// TIA Portal V19 export
ORGANIZATION_BLOCK "MODBUS VFD"   // OB30, LAD, CyclicInterrupt
{ S7_Optimized_Access := 'TRUE' }
// stored: SetENOAutomatically false
   VAR_INPUT
      Initial_Call : Bool;   // Initial call of this OB
      Event_Count : Int;   // Events discarded
   END_VAR
   VAR_TEMP   // added for the SCL form of the ladder/FBD networks
      _w1 : Bool;
      _w2 : Bool;
   END_VAR
BEGIN

REGION Network 2: Slave 1 (SLAVE ID :- 1) WRITE
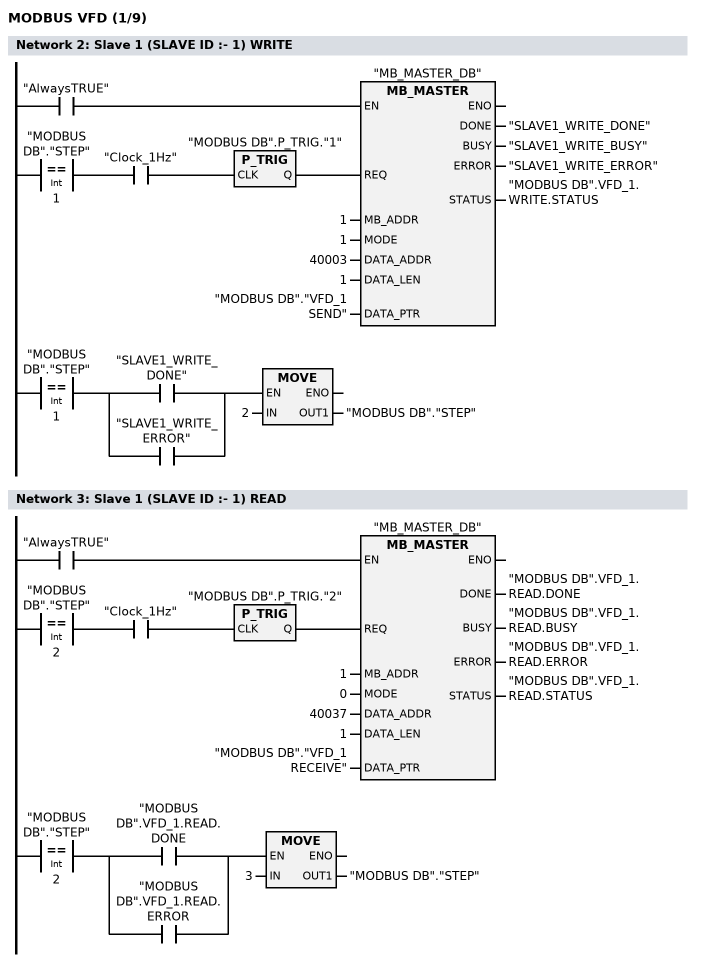
   RUNG wire#powerrail
      Contact( "AlwaysTRUE" )
      "MB_MASTER_DB".MB_MASTER(REQ := wire#w1, MB_ADDR := 1, MODE := 1, DATA_ADDR := 40003, DATA_LEN := 1, DATA_PTR := "MODBUS DB"."VFD_1 SEND", DONE => "SLAVE1_WRITE_DONE", BUSY => "SLAVE1_WRITE_BUSY", ERROR => "SLAVE1_WRITE_ERROR", STATUS => "MODBUS DB".VFD_1.WRITE.STATUS)
   END_RUNG
   RUNG wire#powerrail
      { S7_Templates := "SrcType := Int" } EQ_Contact(in1 := "MODBUS DB"."STEP", in2 := 1)
      Contact( "Clock_1Hz" )
      P_Trig( "MODBUS DB".P_TRIG."1" )
   END_RUNG wire#w1
   RUNG wire#powerrail
      { S7_Templates := "SrcType := Int" } EQ_Contact(in1 := "MODBUS DB"."STEP", in2 := 1)
      wire#w2
      Contact( "SLAVE1_WRITE_DONE" )
      wire#w3
      Move(in := 2, out1 => "MODBUS DB"."STEP")
   END_RUNG
   RUNG wire#w2
      Contact( "SLAVE1_WRITE_ERROR" )
   END_RUNG wire#w3
   // the same network as SCL:
   #_w1 := ("MODBUS DB"."STEP" = 1) AND "Clock_1Hz";
   #_w2 := #_w1 AND NOT "MODBUS DB".P_TRIG."1";   // rising edge
   "MODBUS DB".P_TRIG."1" := #_w1;
   IF "AlwaysTRUE" THEN
       "MB_MASTER_DB"(REQ := #_w2,   // MB_MASTER
                      MB_ADDR := 1,
                      MODE := 1,
                      DATA_ADDR := 40003,
                      DATA_LEN := 1,
                      DATA_PTR := "MODBUS DB"."VFD_1 SEND",
                      DONE => "SLAVE1_WRITE_DONE",
                      BUSY => "SLAVE1_WRITE_BUSY",
                      ERROR => "SLAVE1_WRITE_ERROR",
                      STATUS => "MODBUS DB".VFD_1.WRITE.STATUS);
   END_IF;
   IF ("MODBUS DB"."STEP" = 1) AND ("SLAVE1_WRITE_DONE" OR "SLAVE1_WRITE_ERROR") THEN
       "MODBUS DB"."STEP" := 2;
   END_IF;
END_REGION

REGION Network 3: Slave 1 (SLAVE ID :- 1) READ
   RUNG wire#powerrail
      Contact( "AlwaysTRUE" )
      "MB_MASTER_DB".MB_MASTER(REQ := wire#w1, MB_ADDR := 1, MODE := 0, DATA_ADDR := 40037, DATA_LEN := 1, DATA_PTR := "MODBUS DB"."VFD_1 RECEIVE", DONE => "MODBUS DB".VFD_1.READ.DONE, BUSY => "MODBUS DB".VFD_1.READ.BUSY, ERROR => "MODBUS DB".VFD_1.READ.ERROR, STATUS => "MODBUS DB".VFD_1.READ.STATUS)
   END_RUNG
   RUNG wire#powerrail
      { S7_Templates := "SrcType := Int" } EQ_Contact(in1 := "MODBUS DB"."STEP", in2 := 2)
      Contact( "Clock_1Hz" )
      P_Trig( "MODBUS DB".P_TRIG."2" )
   END_RUNG wire#w1
   RUNG wire#powerrail
      { S7_Templates := "SrcType := Int" } EQ_Contact(in1 := "MODBUS DB"."STEP", in2 := 2)
      wire#w2
      Contact( "MODBUS DB".VFD_1.READ.DONE )
      wire#w3
      Move(in := 3, out1 => "MODBUS DB"."STEP")
   END_RUNG
   RUNG wire#w2
      Contact( "MODBUS DB".VFD_1.READ.ERROR )
   END_RUNG wire#w3
   // the same network as SCL:
   #_w1 := ("MODBUS DB"."STEP" = 2) AND "Clock_1Hz";
   #_w2 := #_w1 AND NOT "MODBUS DB".P_TRIG."2";   // rising edge
   "MODBUS DB".P_TRIG."2" := #_w1;
   IF "AlwaysTRUE" THEN
       "MB_MASTER_DB"(REQ := #_w2,   // MB_MASTER
                      MB_ADDR := 1,
                      MODE := 0,
                      DATA_ADDR := 40037,
                      DATA_LEN := 1,
                      DATA_PTR := "MODBUS DB"."VFD_1 RECEIVE",
                      DONE => "MODBUS DB".VFD_1.READ.DONE,
                      BUSY => "MODBUS DB".VFD_1.READ.BUSY,
                      ERROR => "MODBUS DB".VFD_1.READ.ERROR,
                      STATUS => "MODBUS DB".VFD_1.READ.STATUS);
   END_IF;
   IF ("MODBUS DB"."STEP" = 2) AND ("MODBUS DB".VFD_1.READ.DONE OR "MODBUS DB".VFD_1.READ.ERROR) THEN
       "MODBUS DB"."STEP" := 3;
   END_IF;
END_REGION

REGION Network 4: Slave 2 (SLAVE ID :- 2) WRITE
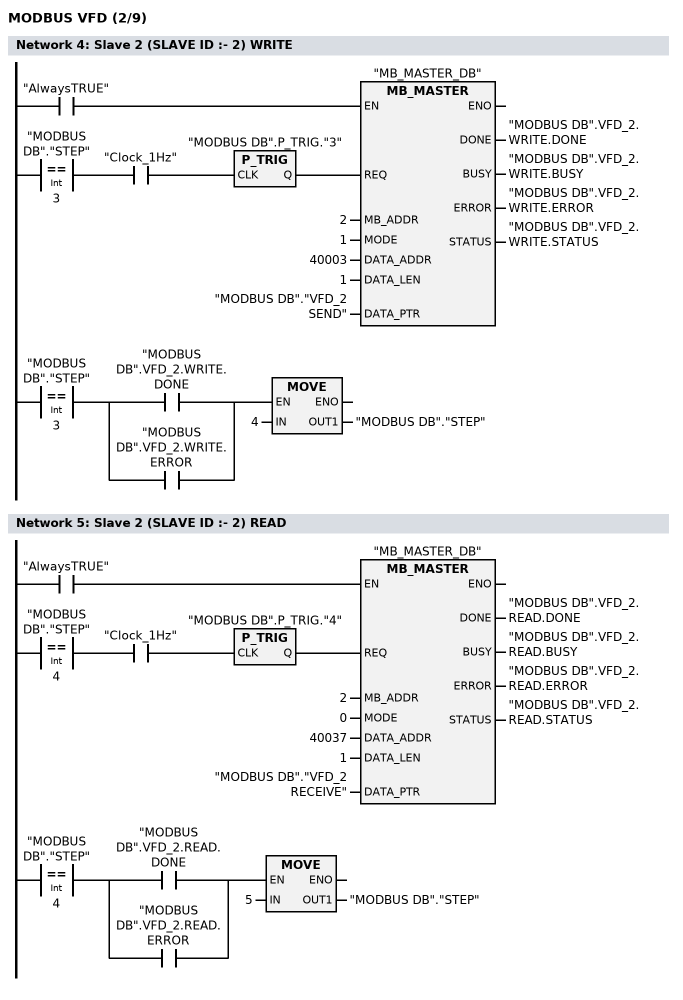
   RUNG wire#powerrail
      Contact( "AlwaysTRUE" )
      "MB_MASTER_DB".MB_MASTER(REQ := wire#w1, MB_ADDR := 2, MODE := 1, DATA_ADDR := 40003, DATA_LEN := 1, DATA_PTR := "MODBUS DB"."VFD_2 SEND", DONE => "MODBUS DB".VFD_2.WRITE.DONE, BUSY => "MODBUS DB".VFD_2.WRITE.BUSY, ERROR => "MODBUS DB".VFD_2.WRITE.ERROR, STATUS => "MODBUS DB".VFD_2.WRITE.STATUS)
   END_RUNG
   RUNG wire#powerrail
      { S7_Templates := "SrcType := Int" } EQ_Contact(in1 := "MODBUS DB"."STEP", in2 := 3)
      Contact( "Clock_1Hz" )
      P_Trig( "MODBUS DB".P_TRIG."3" )
   END_RUNG wire#w1
   RUNG wire#powerrail
      { S7_Templates := "SrcType := Int" } EQ_Contact(in1 := "MODBUS DB"."STEP", in2 := 3)
      wire#w2
      Contact( "MODBUS DB".VFD_2.WRITE.DONE )
      wire#w3
      Move(in := 4, out1 => "MODBUS DB"."STEP")
   END_RUNG
   RUNG wire#w2
      Contact( "MODBUS DB".VFD_2.WRITE.ERROR )
   END_RUNG wire#w3
   // the same network as SCL:
   #_w1 := ("MODBUS DB"."STEP" = 3) AND "Clock_1Hz";
   #_w2 := #_w1 AND NOT "MODBUS DB".P_TRIG."3";   // rising edge
   "MODBUS DB".P_TRIG."3" := #_w1;
   IF "AlwaysTRUE" THEN
       "MB_MASTER_DB"(REQ := #_w2,   // MB_MASTER
                      MB_ADDR := 2,
                      MODE := 1,
                      DATA_ADDR := 40003,
                      DATA_LEN := 1,
                      DATA_PTR := "MODBUS DB"."VFD_2 SEND",
                      DONE => "MODBUS DB".VFD_2.WRITE.DONE,
                      BUSY => "MODBUS DB".VFD_2.WRITE.BUSY,
                      ERROR => "MODBUS DB".VFD_2.WRITE.ERROR,
                      STATUS => "MODBUS DB".VFD_2.WRITE.STATUS);
   END_IF;
   IF ("MODBUS DB"."STEP" = 3) AND ("MODBUS DB".VFD_2.WRITE.DONE OR "MODBUS DB".VFD_2.WRITE.ERROR) THEN
       "MODBUS DB"."STEP" := 4;
   END_IF;
END_REGION

REGION Network 5: Slave 2 (SLAVE ID :- 2) READ
   RUNG wire#powerrail
      Contact( "AlwaysTRUE" )
      "MB_MASTER_DB".MB_MASTER(REQ := wire#w1, MB_ADDR := 2, MODE := 0, DATA_ADDR := 40037, DATA_LEN := 1, DATA_PTR := "MODBUS DB"."VFD_2 RECEIVE", DONE => "MODBUS DB".VFD_2.READ.DONE, BUSY => "MODBUS DB".VFD_2.READ.BUSY, ERROR => "MODBUS DB".VFD_2.READ.ERROR, STATUS => "MODBUS DB".VFD_2.READ.STATUS)
   END_RUNG
   RUNG wire#powerrail
      { S7_Templates := "SrcType := Int" } EQ_Contact(in1 := "MODBUS DB"."STEP", in2 := 4)
      Contact( "Clock_1Hz" )
      P_Trig( "MODBUS DB".P_TRIG."4" )
   END_RUNG wire#w1
   RUNG wire#powerrail
      { S7_Templates := "SrcType := Int" } EQ_Contact(in1 := "MODBUS DB"."STEP", in2 := 4)
      wire#w2
      Contact( "MODBUS DB".VFD_2.READ.DONE )
      wire#w3
      Move(in := 5, out1 => "MODBUS DB"."STEP")
   END_RUNG
   RUNG wire#w2
      Contact( "MODBUS DB".VFD_2.READ.ERROR )
   END_RUNG wire#w3
   // the same network as SCL:
   #_w1 := ("MODBUS DB"."STEP" = 4) AND "Clock_1Hz";
   #_w2 := #_w1 AND NOT "MODBUS DB".P_TRIG."4";   // rising edge
   "MODBUS DB".P_TRIG."4" := #_w1;
   IF "AlwaysTRUE" THEN
       "MB_MASTER_DB"(REQ := #_w2,   // MB_MASTER
                      MB_ADDR := 2,
                      MODE := 0,
                      DATA_ADDR := 40037,
                      DATA_LEN := 1,
                      DATA_PTR := "MODBUS DB"."VFD_2 RECEIVE",
                      DONE => "MODBUS DB".VFD_2.READ.DONE,
                      BUSY => "MODBUS DB".VFD_2.READ.BUSY,
                      ERROR => "MODBUS DB".VFD_2.READ.ERROR,
                      STATUS => "MODBUS DB".VFD_2.READ.STATUS);
   END_IF;
   IF ("MODBUS DB"."STEP" = 4) AND ("MODBUS DB".VFD_2.READ.DONE OR "MODBUS DB".VFD_2.READ.ERROR) THEN
       "MODBUS DB"."STEP" := 5;
   END_IF;
END_REGION

REGION Network 6: Slave 3 (SLAVE ID :- 3) WRITE
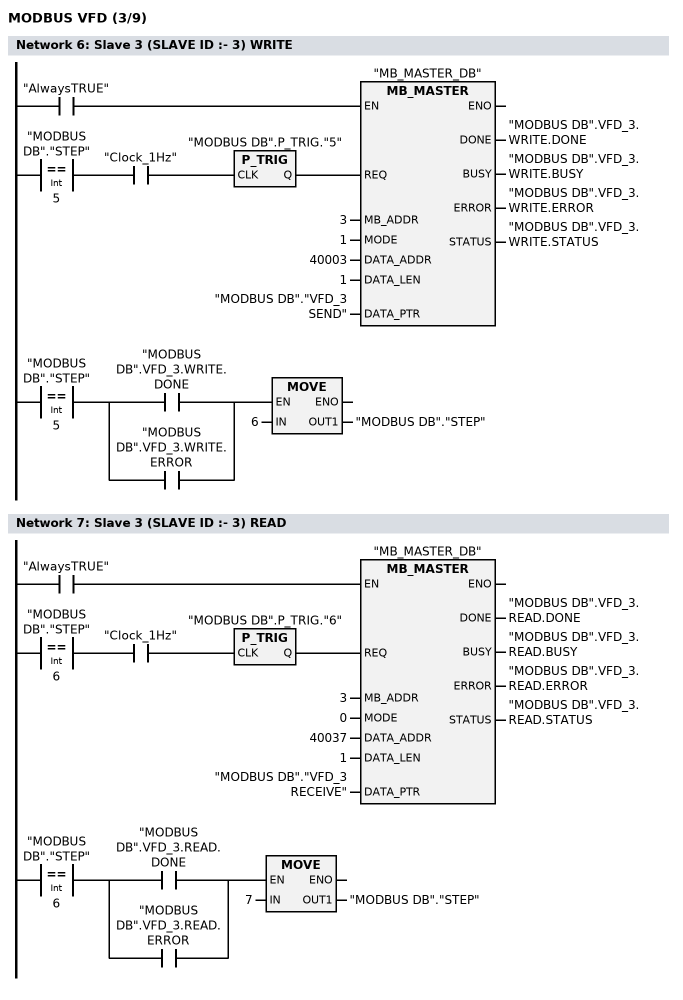
   RUNG wire#powerrail
      Contact( "AlwaysTRUE" )
      "MB_MASTER_DB".MB_MASTER(REQ := wire#w1, MB_ADDR := 3, MODE := 1, DATA_ADDR := 40003, DATA_LEN := 1, DATA_PTR := "MODBUS DB"."VFD_3 SEND", DONE => "MODBUS DB".VFD_3.WRITE.DONE, BUSY => "MODBUS DB".VFD_3.WRITE.BUSY, ERROR => "MODBUS DB".VFD_3.WRITE.ERROR, STATUS => "MODBUS DB".VFD_3.WRITE.STATUS)
   END_RUNG
   RUNG wire#powerrail
      { S7_Templates := "SrcType := Int" } EQ_Contact(in1 := "MODBUS DB"."STEP", in2 := 5)
      Contact( "Clock_1Hz" )
      P_Trig( "MODBUS DB".P_TRIG."5" )
   END_RUNG wire#w1
   RUNG wire#powerrail
      { S7_Templates := "SrcType := Int" } EQ_Contact(in1 := "MODBUS DB"."STEP", in2 := 5)
      wire#w2
      Contact( "MODBUS DB".VFD_3.WRITE.DONE )
      wire#w3
      Move(in := 6, out1 => "MODBUS DB"."STEP")
   END_RUNG
   RUNG wire#w2
      Contact( "MODBUS DB".VFD_3.WRITE.ERROR )
   END_RUNG wire#w3
   // the same network as SCL:
   #_w1 := ("MODBUS DB"."STEP" = 5) AND "Clock_1Hz";
   #_w2 := #_w1 AND NOT "MODBUS DB".P_TRIG."5";   // rising edge
   "MODBUS DB".P_TRIG."5" := #_w1;
   IF "AlwaysTRUE" THEN
       "MB_MASTER_DB"(REQ := #_w2,   // MB_MASTER
                      MB_ADDR := 3,
                      MODE := 1,
                      DATA_ADDR := 40003,
                      DATA_LEN := 1,
                      DATA_PTR := "MODBUS DB"."VFD_3 SEND",
                      DONE => "MODBUS DB".VFD_3.WRITE.DONE,
                      BUSY => "MODBUS DB".VFD_3.WRITE.BUSY,
                      ERROR => "MODBUS DB".VFD_3.WRITE.ERROR,
                      STATUS => "MODBUS DB".VFD_3.WRITE.STATUS);
   END_IF;
   IF ("MODBUS DB"."STEP" = 5) AND ("MODBUS DB".VFD_3.WRITE.DONE OR "MODBUS DB".VFD_3.WRITE.ERROR) THEN
       "MODBUS DB"."STEP" := 6;
   END_IF;
END_REGION

REGION Network 7: Slave 3 (SLAVE ID :- 3) READ
   RUNG wire#powerrail
      Contact( "AlwaysTRUE" )
      "MB_MASTER_DB".MB_MASTER(REQ := wire#w1, MB_ADDR := 3, MODE := 0, DATA_ADDR := 40037, DATA_LEN := 1, DATA_PTR := "MODBUS DB"."VFD_3 RECEIVE", DONE => "MODBUS DB".VFD_3.READ.DONE, BUSY => "MODBUS DB".VFD_3.READ.BUSY, ERROR => "MODBUS DB".VFD_3.READ.ERROR, STATUS => "MODBUS DB".VFD_3.READ.STATUS)
   END_RUNG
   RUNG wire#powerrail
      { S7_Templates := "SrcType := Int" } EQ_Contact(in1 := "MODBUS DB"."STEP", in2 := 6)
      Contact( "Clock_1Hz" )
      P_Trig( "MODBUS DB".P_TRIG."6" )
   END_RUNG wire#w1
   RUNG wire#powerrail
      { S7_Templates := "SrcType := Int" } EQ_Contact(in1 := "MODBUS DB"."STEP", in2 := 6)
      wire#w2
      Contact( "MODBUS DB".VFD_3.READ.DONE )
      wire#w3
      Move(in := 7, out1 => "MODBUS DB"."STEP")
   END_RUNG
   RUNG wire#w2
      Contact( "MODBUS DB".VFD_3.READ.ERROR )
   END_RUNG wire#w3
   // the same network as SCL:
   #_w1 := ("MODBUS DB"."STEP" = 6) AND "Clock_1Hz";
   #_w2 := #_w1 AND NOT "MODBUS DB".P_TRIG."6";   // rising edge
   "MODBUS DB".P_TRIG."6" := #_w1;
   IF "AlwaysTRUE" THEN
       "MB_MASTER_DB"(REQ := #_w2,   // MB_MASTER
                      MB_ADDR := 3,
                      MODE := 0,
                      DATA_ADDR := 40037,
                      DATA_LEN := 1,
                      DATA_PTR := "MODBUS DB"."VFD_3 RECEIVE",
                      DONE => "MODBUS DB".VFD_3.READ.DONE,
                      BUSY => "MODBUS DB".VFD_3.READ.BUSY,
                      ERROR => "MODBUS DB".VFD_3.READ.ERROR,
                      STATUS => "MODBUS DB".VFD_3.READ.STATUS);
   END_IF;
   IF ("MODBUS DB"."STEP" = 6) AND ("MODBUS DB".VFD_3.READ.DONE OR "MODBUS DB".VFD_3.READ.ERROR) THEN
       "MODBUS DB"."STEP" := 7;
   END_IF;
END_REGION

REGION Network 8: Slave 4 (SLAVE ID :- 4) WRITE
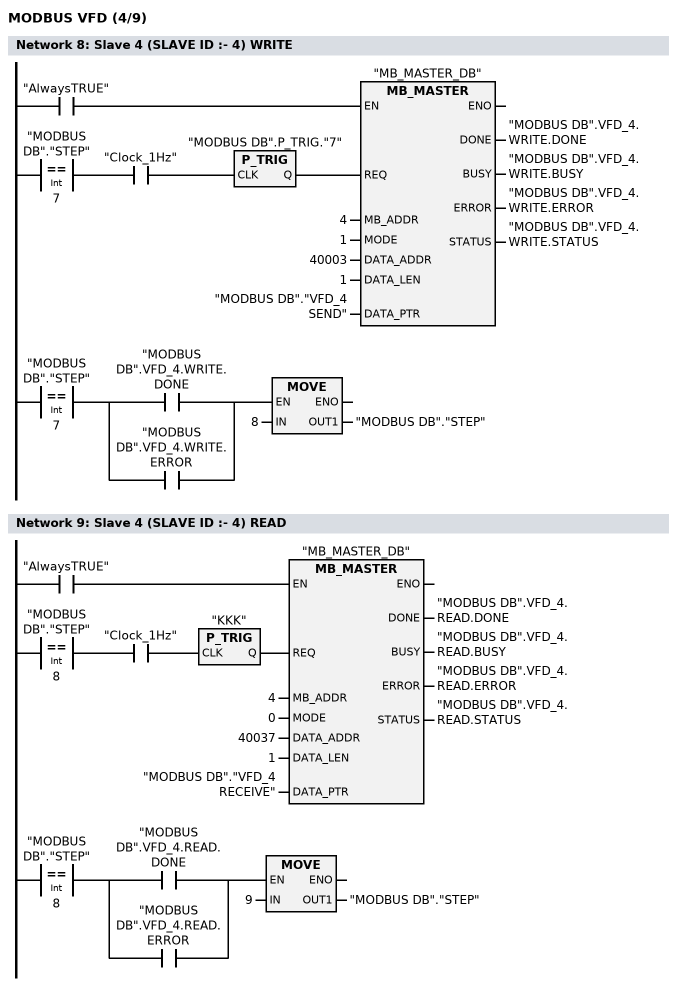
   RUNG wire#powerrail
      Contact( "AlwaysTRUE" )
      "MB_MASTER_DB".MB_MASTER(REQ := wire#w1, MB_ADDR := 4, MODE := 1, DATA_ADDR := 40003, DATA_LEN := 1, DATA_PTR := "MODBUS DB"."VFD_4 SEND", DONE => "MODBUS DB".VFD_4.WRITE.DONE, BUSY => "MODBUS DB".VFD_4.WRITE.BUSY, ERROR => "MODBUS DB".VFD_4.WRITE.ERROR, STATUS => "MODBUS DB".VFD_4.WRITE.STATUS)
   END_RUNG
   RUNG wire#powerrail
      { S7_Templates := "SrcType := Int" } EQ_Contact(in1 := "MODBUS DB"."STEP", in2 := 7)
      Contact( "Clock_1Hz" )
      P_Trig( "MODBUS DB".P_TRIG."7" )
   END_RUNG wire#w1
   RUNG wire#powerrail
      { S7_Templates := "SrcType := Int" } EQ_Contact(in1 := "MODBUS DB"."STEP", in2 := 7)
      wire#w2
      Contact( "MODBUS DB".VFD_4.WRITE.DONE )
      wire#w3
      Move(in := 8, out1 => "MODBUS DB"."STEP")
   END_RUNG
   RUNG wire#w2
      Contact( "MODBUS DB".VFD_4.WRITE.ERROR )
   END_RUNG wire#w3
   // the same network as SCL:
   #_w1 := ("MODBUS DB"."STEP" = 7) AND "Clock_1Hz";
   #_w2 := #_w1 AND NOT "MODBUS DB".P_TRIG."7";   // rising edge
   "MODBUS DB".P_TRIG."7" := #_w1;
   IF "AlwaysTRUE" THEN
       "MB_MASTER_DB"(REQ := #_w2,   // MB_MASTER
                      MB_ADDR := 4,
                      MODE := 1,
                      DATA_ADDR := 40003,
                      DATA_LEN := 1,
                      DATA_PTR := "MODBUS DB"."VFD_4 SEND",
                      DONE => "MODBUS DB".VFD_4.WRITE.DONE,
                      BUSY => "MODBUS DB".VFD_4.WRITE.BUSY,
                      ERROR => "MODBUS DB".VFD_4.WRITE.ERROR,
                      STATUS => "MODBUS DB".VFD_4.WRITE.STATUS);
   END_IF;
   IF ("MODBUS DB"."STEP" = 7) AND ("MODBUS DB".VFD_4.WRITE.DONE OR "MODBUS DB".VFD_4.WRITE.ERROR) THEN
       "MODBUS DB"."STEP" := 8;
   END_IF;
END_REGION

REGION Network 9: Slave 4 (SLAVE ID :- 4) READ
   RUNG wire#powerrail
      Contact( "AlwaysTRUE" )
      "MB_MASTER_DB".MB_MASTER(REQ := wire#w1, MB_ADDR := 4, MODE := 0, DATA_ADDR := 40037, DATA_LEN := 1, DATA_PTR := "MODBUS DB"."VFD_4 RECEIVE", DONE => "MODBUS DB".VFD_4.READ.DONE, BUSY => "MODBUS DB".VFD_4.READ.BUSY, ERROR => "MODBUS DB".VFD_4.READ.ERROR, STATUS => "MODBUS DB".VFD_4.READ.STATUS)
   END_RUNG
   RUNG wire#powerrail
      { S7_Templates := "SrcType := Int" } EQ_Contact(in1 := "MODBUS DB"."STEP", in2 := 8)
      Contact( "Clock_1Hz" )
      P_Trig( "KKK" )
   END_RUNG wire#w1
   RUNG wire#powerrail
      { S7_Templates := "SrcType := Int" } EQ_Contact(in1 := "MODBUS DB"."STEP", in2 := 8)
      wire#w2
      Contact( "MODBUS DB".VFD_4.READ.DONE )
      wire#w3
      Move(in := 9, out1 => "MODBUS DB"."STEP")
   END_RUNG
   RUNG wire#w2
      Contact( "MODBUS DB".VFD_4.READ.ERROR )
   END_RUNG wire#w3
   // the same network as SCL:
   #_w1 := ("MODBUS DB"."STEP" = 8) AND "Clock_1Hz";
   #_w2 := #_w1 AND NOT "KKK";   // rising edge
   "KKK" := #_w1;
   IF "AlwaysTRUE" THEN
       "MB_MASTER_DB"(REQ := #_w2,   // MB_MASTER
                      MB_ADDR := 4,
                      MODE := 0,
                      DATA_ADDR := 40037,
                      DATA_LEN := 1,
                      DATA_PTR := "MODBUS DB"."VFD_4 RECEIVE",
                      DONE => "MODBUS DB".VFD_4.READ.DONE,
                      BUSY => "MODBUS DB".VFD_4.READ.BUSY,
                      ERROR => "MODBUS DB".VFD_4.READ.ERROR,
                      STATUS => "MODBUS DB".VFD_4.READ.STATUS);
   END_IF;
   IF ("MODBUS DB"."STEP" = 8) AND ("MODBUS DB".VFD_4.READ.DONE OR "MODBUS DB".VFD_4.READ.ERROR) THEN
       "MODBUS DB"."STEP" := 9;
   END_IF;
END_REGION

REGION Network 10: Slave 5 (SLAVE ID :- 5) WRITE
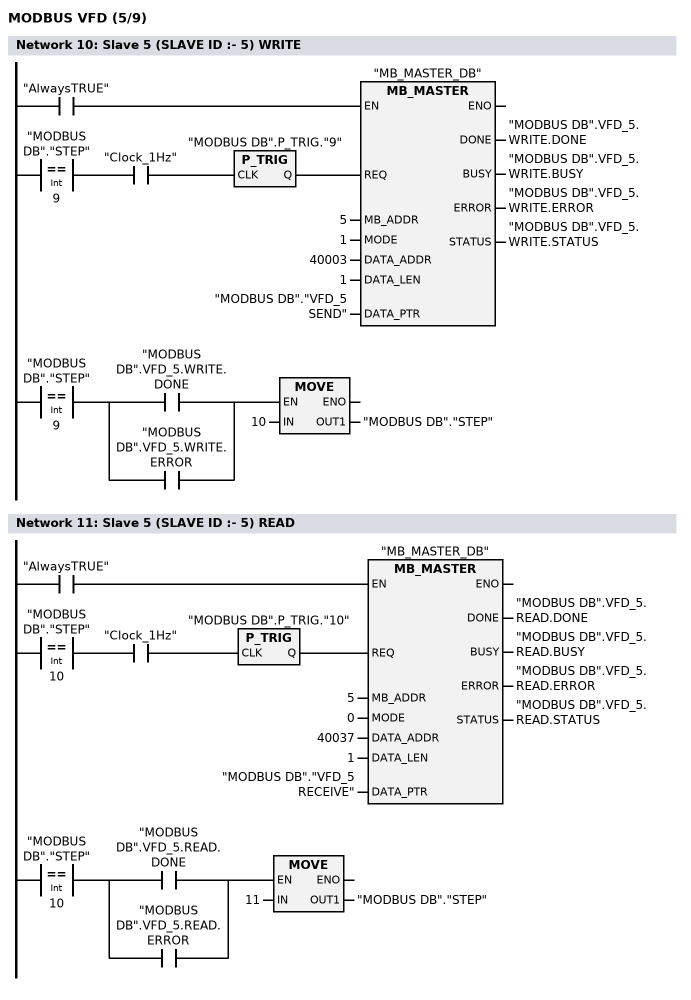
   RUNG wire#powerrail
      Contact( "AlwaysTRUE" )
      "MB_MASTER_DB".MB_MASTER(REQ := wire#w1, MB_ADDR := 5, MODE := 1, DATA_ADDR := 40003, DATA_LEN := 1, DATA_PTR := "MODBUS DB"."VFD_5 SEND", DONE => "MODBUS DB".VFD_5.WRITE.DONE, BUSY => "MODBUS DB".VFD_5.WRITE.BUSY, ERROR => "MODBUS DB".VFD_5.WRITE.ERROR, STATUS => "MODBUS DB".VFD_5.WRITE.STATUS)
   END_RUNG
   RUNG wire#powerrail
      { S7_Templates := "SrcType := Int" } EQ_Contact(in1 := "MODBUS DB"."STEP", in2 := 9)
      Contact( "Clock_1Hz" )
      P_Trig( "MODBUS DB".P_TRIG."9" )
   END_RUNG wire#w1
   RUNG wire#powerrail
      { S7_Templates := "SrcType := Int" } EQ_Contact(in1 := "MODBUS DB"."STEP", in2 := 9)
      wire#w2
      Contact( "MODBUS DB".VFD_5.WRITE.DONE )
      wire#w3
      Move(in := 10, out1 => "MODBUS DB"."STEP")
   END_RUNG
   RUNG wire#w2
      Contact( "MODBUS DB".VFD_5.WRITE.ERROR )
   END_RUNG wire#w3
   // the same network as SCL:
   #_w1 := ("MODBUS DB"."STEP" = 9) AND "Clock_1Hz";
   #_w2 := #_w1 AND NOT "MODBUS DB".P_TRIG."9";   // rising edge
   "MODBUS DB".P_TRIG."9" := #_w1;
   IF "AlwaysTRUE" THEN
       "MB_MASTER_DB"(REQ := #_w2,   // MB_MASTER
                      MB_ADDR := 5,
                      MODE := 1,
                      DATA_ADDR := 40003,
                      DATA_LEN := 1,
                      DATA_PTR := "MODBUS DB"."VFD_5 SEND",
                      DONE => "MODBUS DB".VFD_5.WRITE.DONE,
                      BUSY => "MODBUS DB".VFD_5.WRITE.BUSY,
                      ERROR => "MODBUS DB".VFD_5.WRITE.ERROR,
                      STATUS => "MODBUS DB".VFD_5.WRITE.STATUS);
   END_IF;
   IF ("MODBUS DB"."STEP" = 9) AND ("MODBUS DB".VFD_5.WRITE.DONE OR "MODBUS DB".VFD_5.WRITE.ERROR) THEN
       "MODBUS DB"."STEP" := 10;
   END_IF;
END_REGION

REGION Network 11: Slave 5 (SLAVE ID :- 5) READ
   RUNG wire#powerrail
      Contact( "AlwaysTRUE" )
      "MB_MASTER_DB".MB_MASTER(REQ := wire#w1, MB_ADDR := 5, MODE := 0, DATA_ADDR := 40037, DATA_LEN := 1, DATA_PTR := "MODBUS DB"."VFD_5 RECEIVE", DONE => "MODBUS DB".VFD_5.READ.DONE, BUSY => "MODBUS DB".VFD_5.READ.BUSY, ERROR => "MODBUS DB".VFD_5.READ.ERROR, STATUS => "MODBUS DB".VFD_5.READ.STATUS)
   END_RUNG
   RUNG wire#powerrail
      { S7_Templates := "SrcType := Int" } EQ_Contact(in1 := "MODBUS DB"."STEP", in2 := 10)
      Contact( "Clock_1Hz" )
      P_Trig( "MODBUS DB".P_TRIG."10" )
   END_RUNG wire#w1
   RUNG wire#powerrail
      { S7_Templates := "SrcType := Int" } EQ_Contact(in1 := "MODBUS DB"."STEP", in2 := 10)
      wire#w2
      Contact( "MODBUS DB".VFD_5.READ.DONE )
      wire#w3
      Move(in := 11, out1 => "MODBUS DB"."STEP")
   END_RUNG
   RUNG wire#w2
      Contact( "MODBUS DB".VFD_5.READ.ERROR )
   END_RUNG wire#w3
   // the same network as SCL:
   #_w1 := ("MODBUS DB"."STEP" = 10) AND "Clock_1Hz";
   #_w2 := #_w1 AND NOT "MODBUS DB".P_TRIG."10";   // rising edge
   "MODBUS DB".P_TRIG."10" := #_w1;
   IF "AlwaysTRUE" THEN
       "MB_MASTER_DB"(REQ := #_w2,   // MB_MASTER
                      MB_ADDR := 5,
                      MODE := 0,
                      DATA_ADDR := 40037,
                      DATA_LEN := 1,
                      DATA_PTR := "MODBUS DB"."VFD_5 RECEIVE",
                      DONE => "MODBUS DB".VFD_5.READ.DONE,
                      BUSY => "MODBUS DB".VFD_5.READ.BUSY,
                      ERROR => "MODBUS DB".VFD_5.READ.ERROR,
                      STATUS => "MODBUS DB".VFD_5.READ.STATUS);
   END_IF;
   IF ("MODBUS DB"."STEP" = 10) AND ("MODBUS DB".VFD_5.READ.DONE OR "MODBUS DB".VFD_5.READ.ERROR) THEN
       "MODBUS DB"."STEP" := 11;
   END_IF;
END_REGION

REGION Network 12: Slave 6 (SLAVE ID :- 6) WRITE
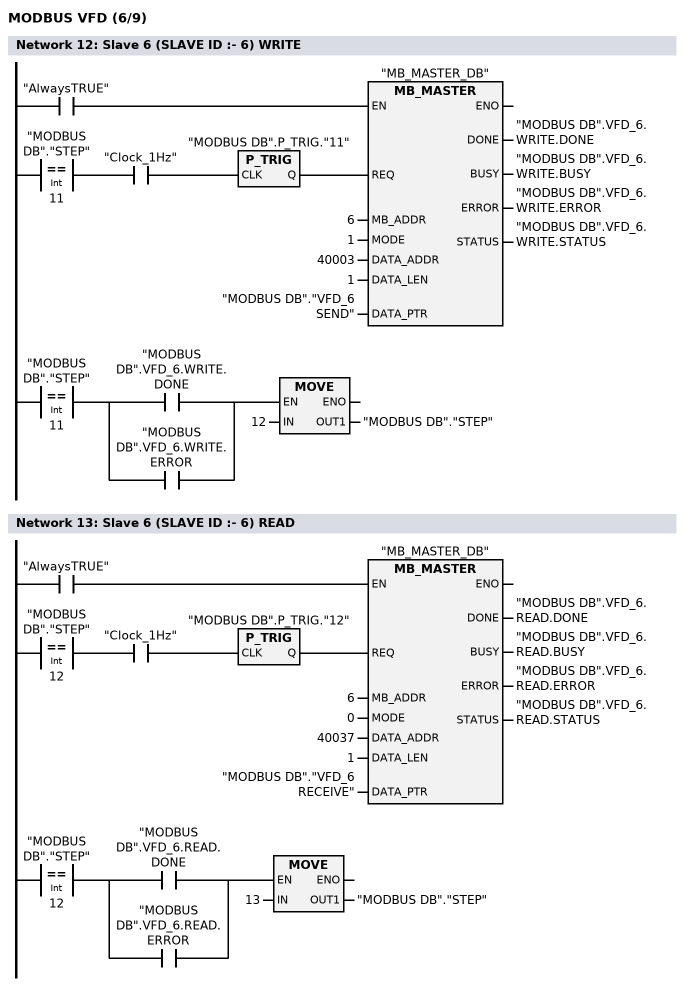
   RUNG wire#powerrail
      Contact( "AlwaysTRUE" )
      "MB_MASTER_DB".MB_MASTER(REQ := wire#w1, MB_ADDR := 6, MODE := 1, DATA_ADDR := 40003, DATA_LEN := 1, DATA_PTR := "MODBUS DB"."VFD_6 SEND", DONE => "MODBUS DB".VFD_6.WRITE.DONE, BUSY => "MODBUS DB".VFD_6.WRITE.BUSY, ERROR => "MODBUS DB".VFD_6.WRITE.ERROR, STATUS => "MODBUS DB".VFD_6.WRITE.STATUS)
   END_RUNG
   RUNG wire#powerrail
      { S7_Templates := "SrcType := Int" } EQ_Contact(in1 := "MODBUS DB"."STEP", in2 := 11)
      Contact( "Clock_1Hz" )
      P_Trig( "MODBUS DB".P_TRIG."11" )
   END_RUNG wire#w1
   RUNG wire#powerrail
      { S7_Templates := "SrcType := Int" } EQ_Contact(in1 := "MODBUS DB"."STEP", in2 := 11)
      wire#w2
      Contact( "MODBUS DB".VFD_6.WRITE.DONE )
      wire#w3
      Move(in := 12, out1 => "MODBUS DB"."STEP")
   END_RUNG
   RUNG wire#w2
      Contact( "MODBUS DB".VFD_6.WRITE.ERROR )
   END_RUNG wire#w3
   // the same network as SCL:
   #_w1 := ("MODBUS DB"."STEP" = 11) AND "Clock_1Hz";
   #_w2 := #_w1 AND NOT "MODBUS DB".P_TRIG."11";   // rising edge
   "MODBUS DB".P_TRIG."11" := #_w1;
   IF "AlwaysTRUE" THEN
       "MB_MASTER_DB"(REQ := #_w2,   // MB_MASTER
                      MB_ADDR := 6,
                      MODE := 1,
                      DATA_ADDR := 40003,
                      DATA_LEN := 1,
                      DATA_PTR := "MODBUS DB"."VFD_6 SEND",
                      DONE => "MODBUS DB".VFD_6.WRITE.DONE,
                      BUSY => "MODBUS DB".VFD_6.WRITE.BUSY,
                      ERROR => "MODBUS DB".VFD_6.WRITE.ERROR,
                      STATUS => "MODBUS DB".VFD_6.WRITE.STATUS);
   END_IF;
   IF ("MODBUS DB"."STEP" = 11) AND ("MODBUS DB".VFD_6.WRITE.DONE OR "MODBUS DB".VFD_6.WRITE.ERROR) THEN
       "MODBUS DB"."STEP" := 12;
   END_IF;
END_REGION

REGION Network 13: Slave 6 (SLAVE ID :- 6) READ
   RUNG wire#powerrail
      Contact( "AlwaysTRUE" )
      "MB_MASTER_DB".MB_MASTER(REQ := wire#w1, MB_ADDR := 6, MODE := 0, DATA_ADDR := 40037, DATA_LEN := 1, DATA_PTR := "MODBUS DB"."VFD_6 RECEIVE", DONE => "MODBUS DB".VFD_6.READ.DONE, BUSY => "MODBUS DB".VFD_6.READ.BUSY, ERROR => "MODBUS DB".VFD_6.READ.ERROR, STATUS => "MODBUS DB".VFD_6.READ.STATUS)
   END_RUNG
   RUNG wire#powerrail
      { S7_Templates := "SrcType := Int" } EQ_Contact(in1 := "MODBUS DB"."STEP", in2 := 12)
      Contact( "Clock_1Hz" )
      P_Trig( "MODBUS DB".P_TRIG."12" )
   END_RUNG wire#w1
   RUNG wire#powerrail
      { S7_Templates := "SrcType := Int" } EQ_Contact(in1 := "MODBUS DB"."STEP", in2 := 12)
      wire#w2
      Contact( "MODBUS DB".VFD_6.READ.DONE )
      wire#w3
      Move(in := 13, out1 => "MODBUS DB"."STEP")
   END_RUNG
   RUNG wire#w2
      Contact( "MODBUS DB".VFD_6.READ.ERROR )
   END_RUNG wire#w3
   // the same network as SCL:
   #_w1 := ("MODBUS DB"."STEP" = 12) AND "Clock_1Hz";
   #_w2 := #_w1 AND NOT "MODBUS DB".P_TRIG."12";   // rising edge
   "MODBUS DB".P_TRIG."12" := #_w1;
   IF "AlwaysTRUE" THEN
       "MB_MASTER_DB"(REQ := #_w2,   // MB_MASTER
                      MB_ADDR := 6,
                      MODE := 0,
                      DATA_ADDR := 40037,
                      DATA_LEN := 1,
                      DATA_PTR := "MODBUS DB"."VFD_6 RECEIVE",
                      DONE => "MODBUS DB".VFD_6.READ.DONE,
                      BUSY => "MODBUS DB".VFD_6.READ.BUSY,
                      ERROR => "MODBUS DB".VFD_6.READ.ERROR,
                      STATUS => "MODBUS DB".VFD_6.READ.STATUS);
   END_IF;
   IF ("MODBUS DB"."STEP" = 12) AND ("MODBUS DB".VFD_6.READ.DONE OR "MODBUS DB".VFD_6.READ.ERROR) THEN
       "MODBUS DB"."STEP" := 13;
   END_IF;
END_REGION

REGION Network 14: Slave 7 (SLAVE ID :- 7) WRITE
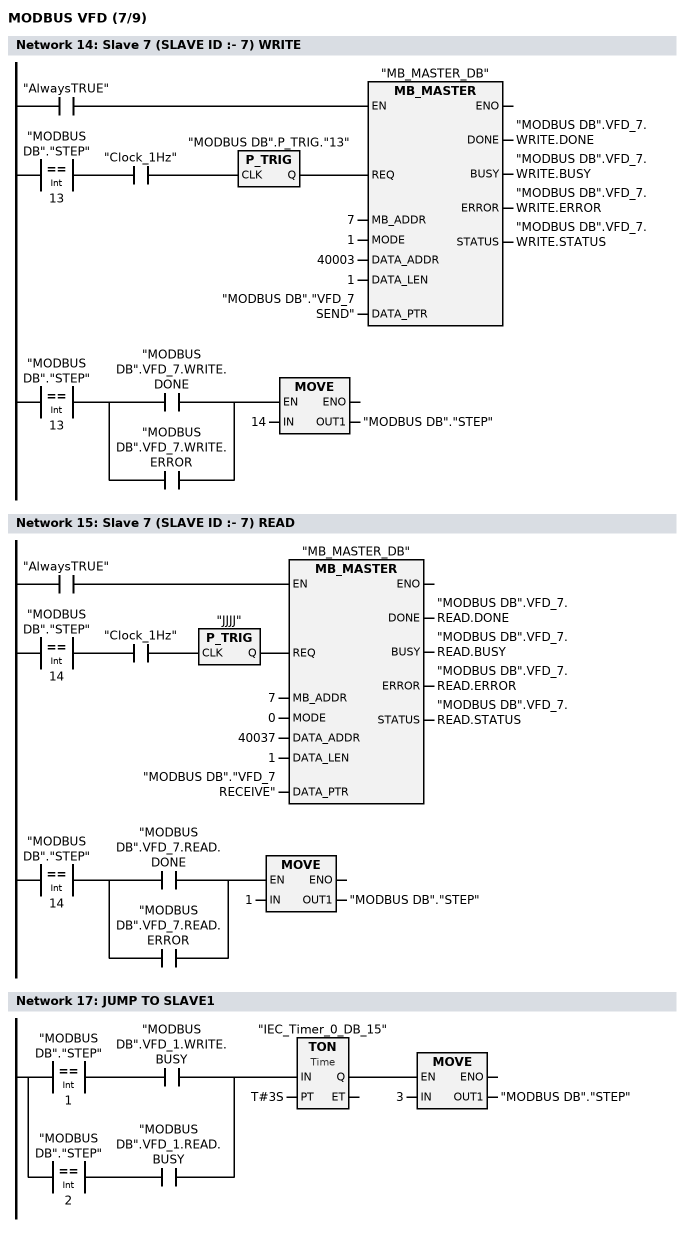
   RUNG wire#powerrail
      Contact( "AlwaysTRUE" )
      "MB_MASTER_DB".MB_MASTER(REQ := wire#w1, MB_ADDR := 7, MODE := 1, DATA_ADDR := 40003, DATA_LEN := 1, DATA_PTR := "MODBUS DB"."VFD_7 SEND", DONE => "MODBUS DB".VFD_7.WRITE.DONE, BUSY => "MODBUS DB".VFD_7.WRITE.BUSY, ERROR => "MODBUS DB".VFD_7.WRITE.ERROR, STATUS => "MODBUS DB".VFD_7.WRITE.STATUS)
   END_RUNG
   RUNG wire#powerrail
      { S7_Templates := "SrcType := Int" } EQ_Contact(in1 := "MODBUS DB"."STEP", in2 := 13)
      Contact( "Clock_1Hz" )
      P_Trig( "MODBUS DB".P_TRIG."13" )
   END_RUNG wire#w1
   RUNG wire#powerrail
      { S7_Templates := "SrcType := Int" } EQ_Contact(in1 := "MODBUS DB"."STEP", in2 := 13)
      wire#w2
      Contact( "MODBUS DB".VFD_7.WRITE.DONE )
      wire#w3
      Move(in := 14, out1 => "MODBUS DB"."STEP")
   END_RUNG
   RUNG wire#w2
      Contact( "MODBUS DB".VFD_7.WRITE.ERROR )
   END_RUNG wire#w3
   // the same network as SCL:
   #_w1 := ("MODBUS DB"."STEP" = 13) AND "Clock_1Hz";
   #_w2 := #_w1 AND NOT "MODBUS DB".P_TRIG."13";   // rising edge
   "MODBUS DB".P_TRIG."13" := #_w1;
   IF "AlwaysTRUE" THEN
       "MB_MASTER_DB"(REQ := #_w2,   // MB_MASTER
                      MB_ADDR := 7,
                      MODE := 1,
                      DATA_ADDR := 40003,
                      DATA_LEN := 1,
                      DATA_PTR := "MODBUS DB"."VFD_7 SEND",
                      DONE => "MODBUS DB".VFD_7.WRITE.DONE,
                      BUSY => "MODBUS DB".VFD_7.WRITE.BUSY,
                      ERROR => "MODBUS DB".VFD_7.WRITE.ERROR,
                      STATUS => "MODBUS DB".VFD_7.WRITE.STATUS);
   END_IF;
   IF ("MODBUS DB"."STEP" = 13) AND ("MODBUS DB".VFD_7.WRITE.DONE OR "MODBUS DB".VFD_7.WRITE.ERROR) THEN
       "MODBUS DB"."STEP" := 14;
   END_IF;
END_REGION

REGION Network 15: Slave 7 (SLAVE ID :- 7) READ
   RUNG wire#powerrail
      Contact( "AlwaysTRUE" )
      "MB_MASTER_DB".MB_MASTER(REQ := wire#w1, MB_ADDR := 7, MODE := 0, DATA_ADDR := 40037, DATA_LEN := 1, DATA_PTR := "MODBUS DB"."VFD_7 RECEIVE", DONE => "MODBUS DB".VFD_7.READ.DONE, BUSY => "MODBUS DB".VFD_7.READ.BUSY, ERROR => "MODBUS DB".VFD_7.READ.ERROR, STATUS => "MODBUS DB".VFD_7.READ.STATUS)
   END_RUNG
   RUNG wire#powerrail
      { S7_Templates := "SrcType := Int" } EQ_Contact(in1 := "MODBUS DB"."STEP", in2 := 14)
      Contact( "Clock_1Hz" )
      P_Trig( "JJJJ" )
   END_RUNG wire#w1
   RUNG wire#powerrail
      { S7_Templates := "SrcType := Int" } EQ_Contact(in1 := "MODBUS DB"."STEP", in2 := 14)
      wire#w2
      Contact( "MODBUS DB".VFD_7.READ.DONE )
      wire#w3
      Move(in := 1, out1 => "MODBUS DB"."STEP")
   END_RUNG
   RUNG wire#w2
      Contact( "MODBUS DB".VFD_7.READ.ERROR )
   END_RUNG wire#w3
   // the same network as SCL:
   #_w1 := ("MODBUS DB"."STEP" = 14) AND "Clock_1Hz";
   #_w2 := #_w1 AND NOT "JJJJ";   // rising edge
   "JJJJ" := #_w1;
   IF "AlwaysTRUE" THEN
       "MB_MASTER_DB"(REQ := #_w2,   // MB_MASTER
                      MB_ADDR := 7,
                      MODE := 0,
                      DATA_ADDR := 40037,
                      DATA_LEN := 1,
                      DATA_PTR := "MODBUS DB"."VFD_7 RECEIVE",
                      DONE => "MODBUS DB".VFD_7.READ.DONE,
                      BUSY => "MODBUS DB".VFD_7.READ.BUSY,
                      ERROR => "MODBUS DB".VFD_7.READ.ERROR,
                      STATUS => "MODBUS DB".VFD_7.READ.STATUS);
   END_IF;
   IF ("MODBUS DB"."STEP" = 14) AND ("MODBUS DB".VFD_7.READ.DONE OR "MODBUS DB".VFD_7.READ.ERROR) THEN
       "MODBUS DB"."STEP" := 1;
   END_IF;
END_REGION

REGION Network 17: JUMP TO SLAVE1
   RUNG wire#powerrail
      { S7_Templates := "SrcType := Int" } EQ_Contact(in1 := "MODBUS DB"."STEP", in2 := 1)
      Contact( "MODBUS DB".VFD_1.WRITE.BUSY )
      wire#w1
      { S7_Templates := "time_type := Time" } "IEC_Timer_0_DB_15".TON(pt := T#3S, et =>)
      Move(in := 3, out1 => "MODBUS DB"."STEP")
   END_RUNG
   RUNG wire#powerrail
      { S7_Templates := "SrcType := Int" } EQ_Contact(in1 := "MODBUS DB"."STEP", in2 := 2)
      Contact( "MODBUS DB".VFD_1.READ.BUSY )
   END_RUNG wire#w1
   // the same network as SCL:
   "IEC_Timer_0_DB_15".TON(IN := (("MODBUS DB"."STEP" = 1) AND "MODBUS DB".VFD_1.WRITE.BUSY) OR (("MODBUS DB"."STEP" = 2) AND "MODBUS DB".VFD_1.READ.BUSY),
                           PT := T#3S);
   IF "IEC_Timer_0_DB_15".Q THEN "MODBUS DB"."STEP" := 3; END_IF;
END_REGION

REGION Network 18: JUMP TO SLAVE2
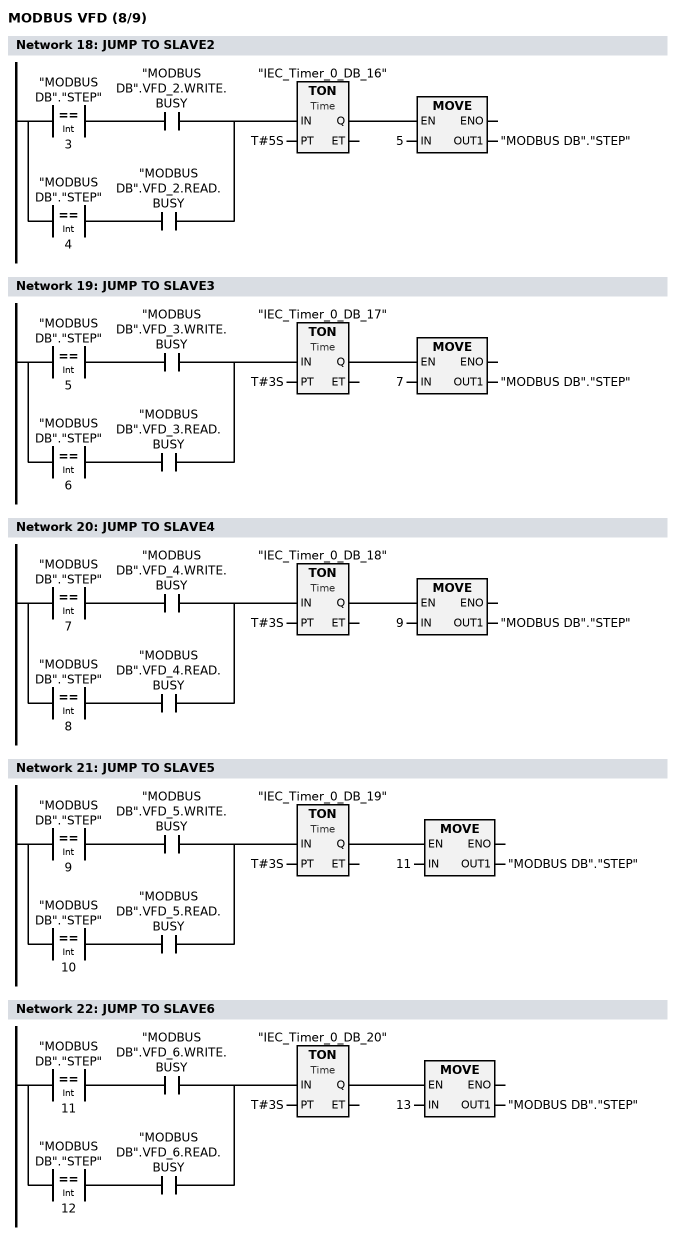
   RUNG wire#powerrail
      { S7_Templates := "SrcType := Int" } EQ_Contact(in1 := "MODBUS DB"."STEP", in2 := 3)
      Contact( "MODBUS DB".VFD_2.WRITE.BUSY )
      wire#w1
      { S7_Templates := "time_type := Time" } "IEC_Timer_0_DB_16".TON(pt := T#5S, et =>)
      Move(in := 5, out1 => "MODBUS DB"."STEP")
   END_RUNG
   RUNG wire#powerrail
      { S7_Templates := "SrcType := Int" } EQ_Contact(in1 := "MODBUS DB"."STEP", in2 := 4)
      Contact( "MODBUS DB".VFD_2.READ.BUSY )
   END_RUNG wire#w1
   // the same network as SCL:
   "IEC_Timer_0_DB_16".TON(IN := (("MODBUS DB"."STEP" = 3) AND "MODBUS DB".VFD_2.WRITE.BUSY) OR (("MODBUS DB"."STEP" = 4) AND "MODBUS DB".VFD_2.READ.BUSY),
                           PT := T#5S);
   IF "IEC_Timer_0_DB_16".Q THEN "MODBUS DB"."STEP" := 5; END_IF;
END_REGION

REGION Network 19: JUMP TO SLAVE3
   RUNG wire#powerrail
      { S7_Templates := "SrcType := Int" } EQ_Contact(in1 := "MODBUS DB"."STEP", in2 := 5)
      Contact( "MODBUS DB".VFD_3.WRITE.BUSY )
      wire#w1
      { S7_Templates := "time_type := Time" } "IEC_Timer_0_DB_17".TON(pt := T#3S, et =>)
      Move(in := 7, out1 => "MODBUS DB"."STEP")
   END_RUNG
   RUNG wire#powerrail
      { S7_Templates := "SrcType := Int" } EQ_Contact(in1 := "MODBUS DB"."STEP", in2 := 6)
      Contact( "MODBUS DB".VFD_3.READ.BUSY )
   END_RUNG wire#w1
   // the same network as SCL:
   "IEC_Timer_0_DB_17".TON(IN := (("MODBUS DB"."STEP" = 5) AND "MODBUS DB".VFD_3.WRITE.BUSY) OR (("MODBUS DB"."STEP" = 6) AND "MODBUS DB".VFD_3.READ.BUSY),
                           PT := T#3S);
   IF "IEC_Timer_0_DB_17".Q THEN "MODBUS DB"."STEP" := 7; END_IF;
END_REGION

REGION Network 20: JUMP TO SLAVE4
   RUNG wire#powerrail
      { S7_Templates := "SrcType := Int" } EQ_Contact(in1 := "MODBUS DB"."STEP", in2 := 7)
      Contact( "MODBUS DB".VFD_4.WRITE.BUSY )
      wire#w1
      { S7_Templates := "time_type := Time" } "IEC_Timer_0_DB_18".TON(pt := T#3S, et =>)
      Move(in := 9, out1 => "MODBUS DB"."STEP")
   END_RUNG
   RUNG wire#powerrail
      { S7_Templates := "SrcType := Int" } EQ_Contact(in1 := "MODBUS DB"."STEP", in2 := 8)
      Contact( "MODBUS DB".VFD_4.READ.BUSY )
   END_RUNG wire#w1
   // the same network as SCL:
   "IEC_Timer_0_DB_18".TON(IN := (("MODBUS DB"."STEP" = 7) AND "MODBUS DB".VFD_4.WRITE.BUSY) OR (("MODBUS DB"."STEP" = 8) AND "MODBUS DB".VFD_4.READ.BUSY),
                           PT := T#3S);
   IF "IEC_Timer_0_DB_18".Q THEN "MODBUS DB"."STEP" := 9; END_IF;
END_REGION

REGION Network 21: JUMP TO SLAVE5
   RUNG wire#powerrail
      { S7_Templates := "SrcType := Int" } EQ_Contact(in1 := "MODBUS DB"."STEP", in2 := 9)
      Contact( "MODBUS DB".VFD_5.WRITE.BUSY )
      wire#w1
      { S7_Templates := "time_type := Time" } "IEC_Timer_0_DB_19".TON(pt := T#3S, et =>)
      Move(in := 11, out1 => "MODBUS DB"."STEP")
   END_RUNG
   RUNG wire#powerrail
      { S7_Templates := "SrcType := Int" } EQ_Contact(in1 := "MODBUS DB"."STEP", in2 := 10)
      Contact( "MODBUS DB".VFD_5.READ.BUSY )
   END_RUNG wire#w1
   // the same network as SCL:
   "IEC_Timer_0_DB_19".TON(IN := (("MODBUS DB"."STEP" = 9) AND "MODBUS DB".VFD_5.WRITE.BUSY) OR (("MODBUS DB"."STEP" = 10) AND "MODBUS DB".VFD_5.READ.BUSY),
                           PT := T#3S);
   IF "IEC_Timer_0_DB_19".Q THEN "MODBUS DB"."STEP" := 11; END_IF;
END_REGION

REGION Network 22: JUMP TO SLAVE6
   RUNG wire#powerrail
      { S7_Templates := "SrcType := Int" } EQ_Contact(in1 := "MODBUS DB"."STEP", in2 := 11)
      Contact( "MODBUS DB".VFD_6.WRITE.BUSY )
      wire#w1
      { S7_Templates := "time_type := Time" } "IEC_Timer_0_DB_20".TON(pt := T#3S, et =>)
      Move(in := 13, out1 => "MODBUS DB"."STEP")
   END_RUNG
   RUNG wire#powerrail
      { S7_Templates := "SrcType := Int" } EQ_Contact(in1 := "MODBUS DB"."STEP", in2 := 12)
      Contact( "MODBUS DB".VFD_6.READ.BUSY )
   END_RUNG wire#w1
   // the same network as SCL:
   "IEC_Timer_0_DB_20".TON(IN := (("MODBUS DB"."STEP" = 11) AND "MODBUS DB".VFD_6.WRITE.BUSY) OR (("MODBUS DB"."STEP" = 12) AND "MODBUS DB".VFD_6.READ.BUSY),
                           PT := T#3S);
   IF "IEC_Timer_0_DB_20".Q THEN "MODBUS DB"."STEP" := 13; END_IF;
END_REGION

REGION Network 23: JUMP TO SLAVE7
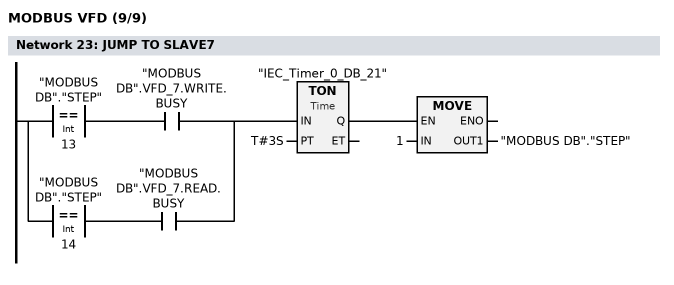
   RUNG wire#powerrail
      { S7_Templates := "SrcType := Int" } EQ_Contact(in1 := "MODBUS DB"."STEP", in2 := 13)
      Contact( "MODBUS DB".VFD_7.WRITE.BUSY )
      wire#w1
      { S7_Templates := "time_type := Time" } "IEC_Timer_0_DB_21".TON(pt := T#3S, et =>)
      Move(in := 1, out1 => "MODBUS DB"."STEP")
   END_RUNG
   RUNG wire#powerrail
      { S7_Templates := "SrcType := Int" } EQ_Contact(in1 := "MODBUS DB"."STEP", in2 := 14)
      Contact( "MODBUS DB".VFD_7.READ.BUSY )
   END_RUNG wire#w1
   // the same network as SCL:
   "IEC_Timer_0_DB_21".TON(IN := (("MODBUS DB"."STEP" = 13) AND "MODBUS DB".VFD_7.WRITE.BUSY) OR (("MODBUS DB"."STEP" = 14) AND "MODBUS DB".VFD_7.READ.BUSY),
                           PT := T#3S);
   IF "IEC_Timer_0_DB_21".Q THEN "MODBUS DB"."STEP" := 1; END_IF;
END_REGION
END_ORGANIZATION_BLOCK
